{attribute 'qualified_only'}
{attribute 'strict'}
TYPE eInstalState :
(
	InProgress := 0,
	Success	   := 1,
	Failure	   := 2
);
END_TYPE

(* stored: Version 1.1.0.1, ProductVersion 3.1.4026.18
   DUT eInstalState: Id {63734c68-e75b-4487-a132-0cf19f1732a1} *)
